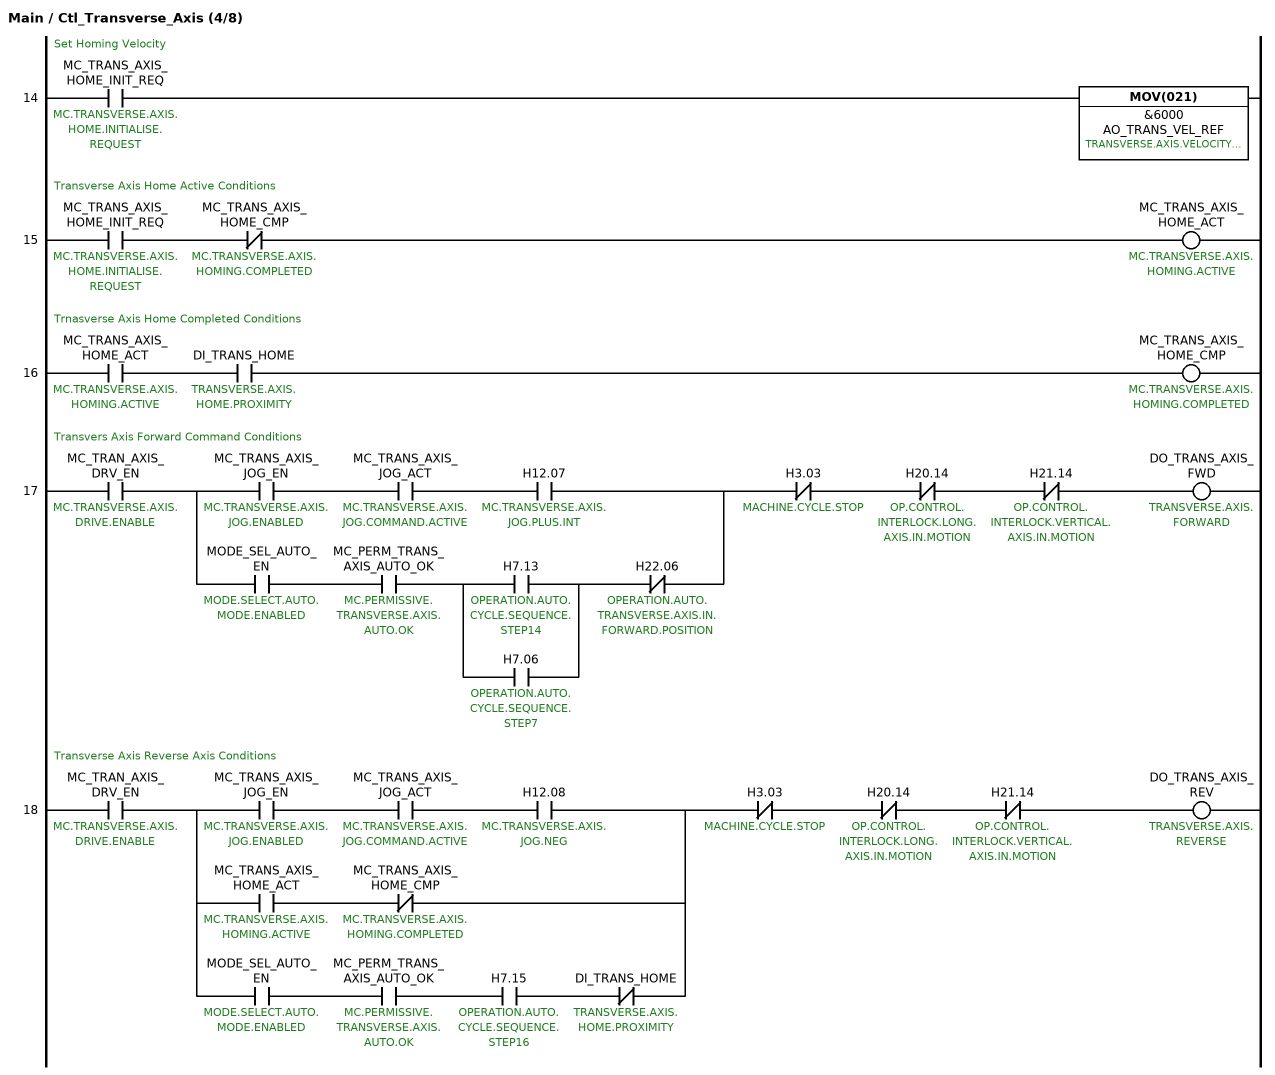
; [picture p48: Main / Ctl_Transverse_Axis, rungs 14-18]
; rung 14: Set Homing Velocity
LD MC_TRANS_AXIS_HOME_INIT_REQ  ; MC.TRANSVERSE.AXIS.HOME.INITIALISE.REQUEST
MOV(021) &6000 AO_TRANS_VEL_REF  ; TRANSVERSE.AXIS.VELOCITY.ANALOG.REFERENCE
; rung 15: Transverse Axis Home Active Conditions
LD MC_TRANS_AXIS_HOME_INIT_REQ  ; MC.TRANSVERSE.AXIS.HOME.INITIALISE.REQUEST
ANDNOT MC_TRANS_AXIS_HOME_CMP  ; MC.TRANSVERSE.AXIS.HOMING.COMPLETED
OUT MC_TRANS_AXIS_HOME_ACT  ; MC.TRANSVERSE.AXIS.HOMING.ACTIVE
; rung 16: Trnasverse Axis Home Completed Conditions
LD MC_TRANS_AXIS_HOME_ACT  ; MC.TRANSVERSE.AXIS.HOMING.ACTIVE
AND DI_TRANS_HOME  ; TRANSVERSE.AXIS.HOME.PROXIMITY
OUT MC_TRANS_AXIS_HOME_CMP  ; MC.TRANSVERSE.AXIS.HOMING.COMPLETED
; rung 17: Transvers Axis Forward Command Conditions
LD MC_TRAN_AXIS_DRV_EN  ; MC.TRANSVERSE.AXIS.DRIVE.ENABLE
LD MC_TRANS_AXIS_JOG_EN  ; MC.TRANSVERSE.AXIS.JOG.ENABLED
AND MC_TRANS_AXIS_JOG_ACT  ; MC.TRANSVERSE.AXIS.JOG.COMMAND.ACTIVE
AND H12.07  ; MC.TRANSVERSE.AXIS.JOG.PLUS.INT
LD MODE_SEL_AUTO_EN  ; MODE.SELECT.AUTO.MODE.ENABLED
AND MC_PERM_TRANS_AXIS_AUTO_OK  ; MC.PERMISSIVE.TRANSVERSE.AXIS.AUTO.OK
LD H7.13  ; OPERATION.AUTO.CYCLE.SEQUENCE.STEP14
OR H7.06  ; OPERATION.AUTO.CYCLE.SEQUENCE.STEP7
ANDLD
ANDNOT H22.06  ; OPERATION.AUTO.TRANSVERSE.AXIS.IN.FORWARD.POSITION
ORLD
ANDLD
ANDNOT H3.03  ; MACHINE.CYCLE.STOP
ANDNOT H20.14  ; OP.CONTROL.INTERLOCK.LONG.AXIS.IN.MOTION
ANDNOT H21.14  ; OP.CONTROL.INTERLOCK.VERTICAL.AXIS.IN.MOTION
OUT DO_TRANS_AXIS_FWD  ; TRANSVERSE.AXIS.FORWARD
; rung 18: Transverse Axis Reverse Axis Conditions
LD MC_TRAN_AXIS_DRV_EN  ; MC.TRANSVERSE.AXIS.DRIVE.ENABLE
LD MC_TRANS_AXIS_JOG_EN  ; MC.TRANSVERSE.AXIS.JOG.ENABLED
AND MC_TRANS_AXIS_JOG_ACT  ; MC.TRANSVERSE.AXIS.JOG.COMMAND.ACTIVE
AND H12.08  ; MC.TRANSVERSE.AXIS.JOG.NEG
LD MC_TRANS_AXIS_HOME_ACT  ; MC.TRANSVERSE.AXIS.HOMING.ACTIVE
ANDNOT MC_TRANS_AXIS_HOME_CMP  ; MC.TRANSVERSE.AXIS.HOMING.COMPLETED
ORLD
LD MODE_SEL_AUTO_EN  ; MODE.SELECT.AUTO.MODE.ENABLED
AND MC_PERM_TRANS_AXIS_AUTO_OK  ; MC.PERMISSIVE.TRANSVERSE.AXIS.AUTO.OK
AND H7.15  ; OPERATION.AUTO.CYCLE.SEQUENCE.STEP16
ANDNOT DI_TRANS_HOME  ; TRANSVERSE.AXIS.HOME.PROXIMITY
ORLD
ANDLD
ANDNOT H3.03  ; MACHINE.CYCLE.STOP
ANDNOT H20.14  ; OP.CONTROL.INTERLOCK.LONG.AXIS.IN.MOTION
ANDNOT H21.14  ; OP.CONTROL.INTERLOCK.VERTICAL.AXIS.IN.MOTION
OUT DO_TRANS_AXIS_REV  ; TRANSVERSE.AXIS.REVERSE

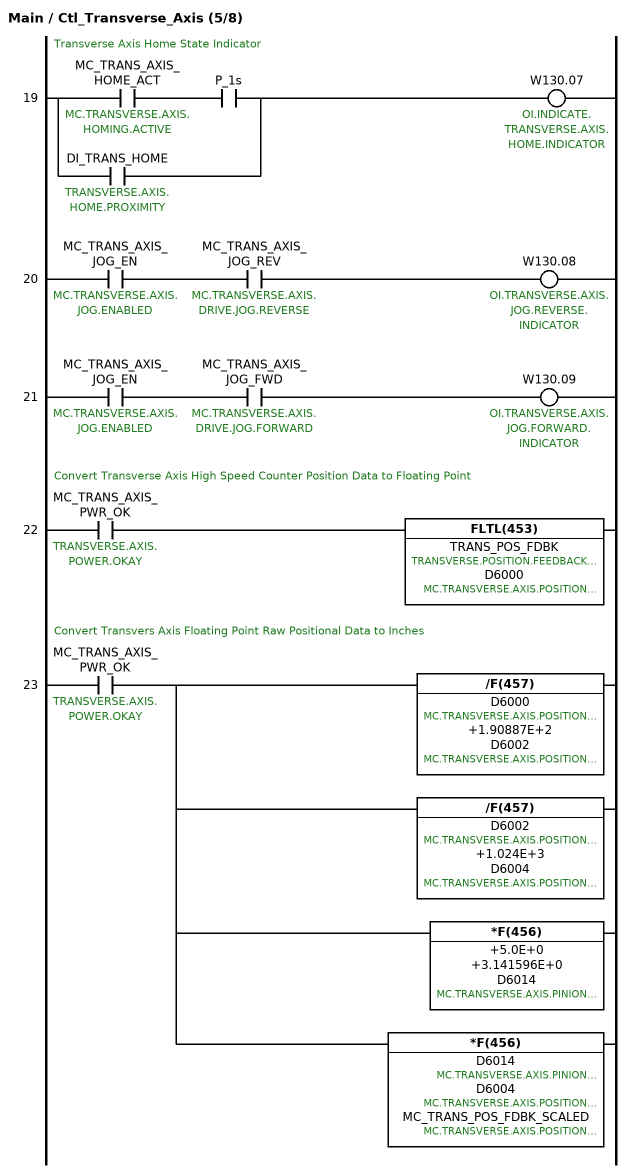
; rung 19: Transverse Axis Home State Indicator
LD MC_TRANS_AXIS_HOME_ACT  ; MC.TRANSVERSE.AXIS.HOMING.ACTIVE
AND P_1s
OR DI_TRANS_HOME  ; TRANSVERSE.AXIS.HOME.PROXIMITY
OUT W130.07  ; OI.INDICATE.TRANSVERSE.AXIS.HOME.INDICATOR
; rung 20
LD MC_TRANS_AXIS_JOG_EN  ; MC.TRANSVERSE.AXIS.JOG.ENABLED
AND MC_TRANS_AXIS_JOG_REV  ; MC.TRANSVERSE.AXIS.DRIVE.JOG.REVERSE
OUT W130.08  ; OI.TRANSVERSE.AXIS.JOG.REVERSE.INDICATOR
; rung 21
LD MC_TRANS_AXIS_JOG_EN  ; MC.TRANSVERSE.AXIS.JOG.ENABLED
AND MC_TRANS_AXIS_JOG_FWD  ; MC.TRANSVERSE.AXIS.DRIVE.JOG.FORWARD
OUT W130.09  ; OI.TRANSVERSE.AXIS.JOG.FORWARD.INDICATOR
; rung 22: Convert Transverse Axis High Speed Counter Position Data to Floating Point
LD MC_TRANS_AXIS_PWR_OK  ; TRANSVERSE.AXIS.POWER.OKAY
FLTL(453) TRANS_POS_FDBK D6000  ; TRANSVERSE.POSITION.FEEDBACK.RAW, MC.TRANSVERSE.AXIS.POSITION.FEEDBACK.RAW.REAL
; rung 23: Convert Transvers Axis Floating Point Raw Positional Data to Inches
LD MC_TRANS_AXIS_PWR_OK  ; TRANSVERSE.AXIS.POWER.OKAY
/F(457) D6000 +1.90887E+2 D6002  ; MC.TRANSVERSE.AXIS.POSITION.FEEDBACK.RAW.REAL, MC.TRANSVERSE.AXIS.POSITION.FEEDBACK.GB.SCALED.REAL
/F(457) D6002 +1.024E+3 D6004  ; MC.TRANSVERSE.AXIS.POSITION.FEEDBACK.GB.SCALED.REAL, MC.TRANSVERSE.AXIS.POSITION.PINION.REVOLUTIONS.REAL
*F(456) +5.0E+0 +3.141596E+0 D6014  ; MC.TRANSVERSE.AXIS.PINION.CIRCUMFERENCE.INCHES.REAL
*F(456) D6014 D6004 MC_TRANS_POS_FDBK_SCALED  ; MC.TRANSVERSE.AXIS.PINION.CIRCUMFERENCE.INCHES.REAL, MC.TRANSVERSE.AXIS.POSITION.PINION.REVOLUTIONS.REAL, MC.TRANSVERSE.AXIS.POSITION.FEEDBACK.INCHES.SCALED.REAL

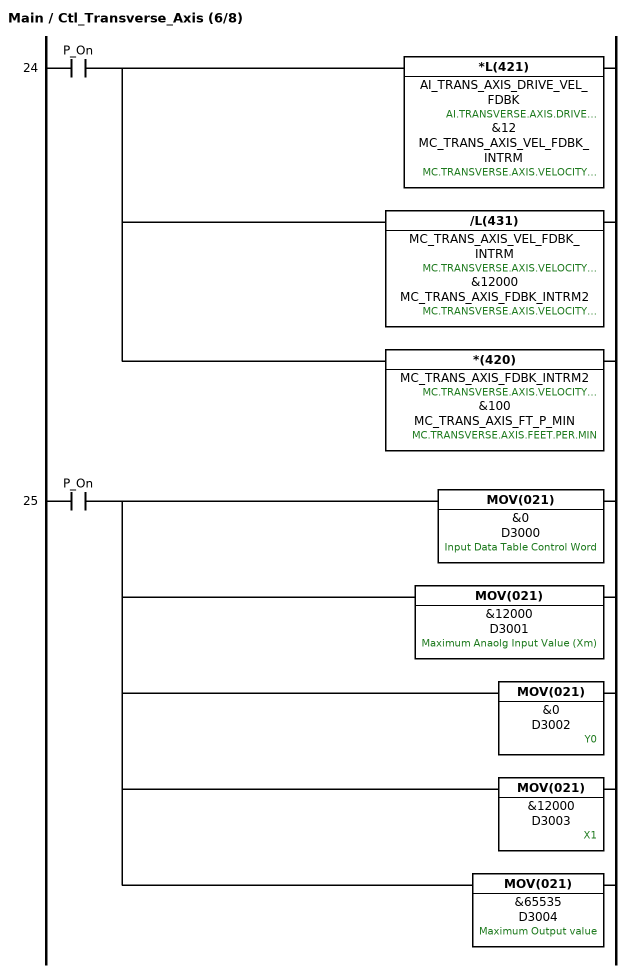
; rung 24
LD P_On
*L(421) AI_TRANS_AXIS_DRIVE_VEL_FDBK &12 MC_TRANS_AXIS_VEL_FDBK_INTRM  ; AI.TRANSVERSE.AXIS.DRIVE.VELOCITY.FEEDBACK, MC.TRANSVERSE.AXIS.VELOCITY.FEEDBACK.INTERIM
/L(431) MC_TRANS_AXIS_VEL_FDBK_INTRM &12000 MC_TRANS_AXIS_FDBK_INTRM2  ; MC.TRANSVERSE.AXIS.VELOCITY.FEEDBACK.INTERIM, MC.TRANSVERSE.AXIS.VELOCITY.FEEDBACK.INTERIM2
*(420) MC_TRANS_AXIS_FDBK_INTRM2 &100 MC_TRANS_AXIS_FT_P_MIN  ; MC.TRANSVERSE.AXIS.VELOCITY.FEEDBACK.INTERIM2, MC.TRANSVERSE.AXIS.FEET.PER.MIN
; rung 25
LD P_On
MOV(021) &0 D3000  ; Input Data Table Control Word
MOV(021) &12000 D3001  ; Maximum Anaolg Input Value (Xm)
MOV(021) &0 D3002  ; Y0
MOV(021) &12000 D3003  ; X1
MOV(021) &65535 D3004  ; Maximum Output value

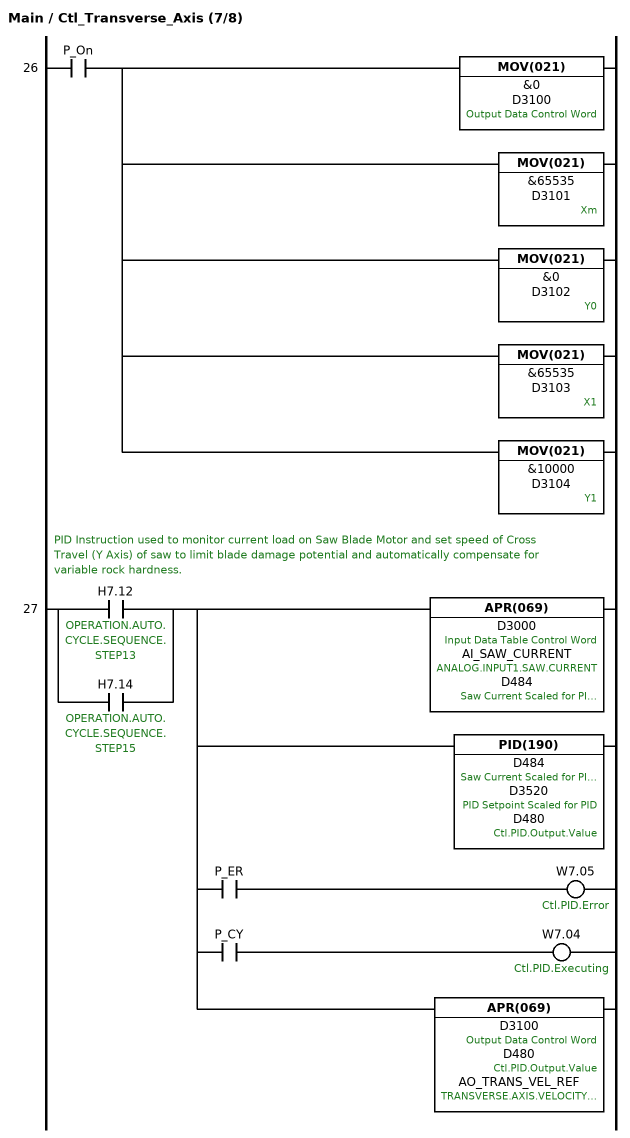
; rung 26
LD P_On
MOV(021) &0 D3100  ; Output Data Control Word
MOV(021) &65535 D3101  ; Xm
MOV(021) &0 D3102  ; Y0
MOV(021) &65535 D3103  ; X1
MOV(021) &10000 D3104  ; Y1
; rung 27: PID Instruction used to monitor current load on Saw Blade Motor and set speed of Cross Travel (Y Axis) of saw to limit blade damage potential and automatically compensate for variable rock hardness.
LD H7.12  ; OPERATION.AUTO.CYCLE.SEQUENCE.STEP13
OR H7.14  ; OPERATION.AUTO.CYCLE.SEQUENCE.STEP15
OUT TR0
APR(069) D3000 AI_SAW_CURRENT D484  ; Input Data Table Control Word, ANALOG.INPUT1.SAW.CURRENT, Saw Current Scaled for PID instruction use
PID(190) D484 D3520 D480  ; Saw Current Scaled for PID instruction use, PID Setpoint Scaled for PID, Ctl.PID.Output.Value
AND P_ER
OUT W7.05  ; Ctl.PID.Error  // Set BitW7.05 to High if PID instruction Errors
LD TR0
AND P_CY
OUT W7.04  ; Ctl.PID.Executing  // When PID is executing W7.04 is High
LD TR0
APR(069) D3100 D480 AO_TRANS_VEL_REF  ; Output Data Control Word, Ctl.PID.Output.Value, TRANSVERSE.AXIS.VELOCITY.ANALOG.REFERENCE

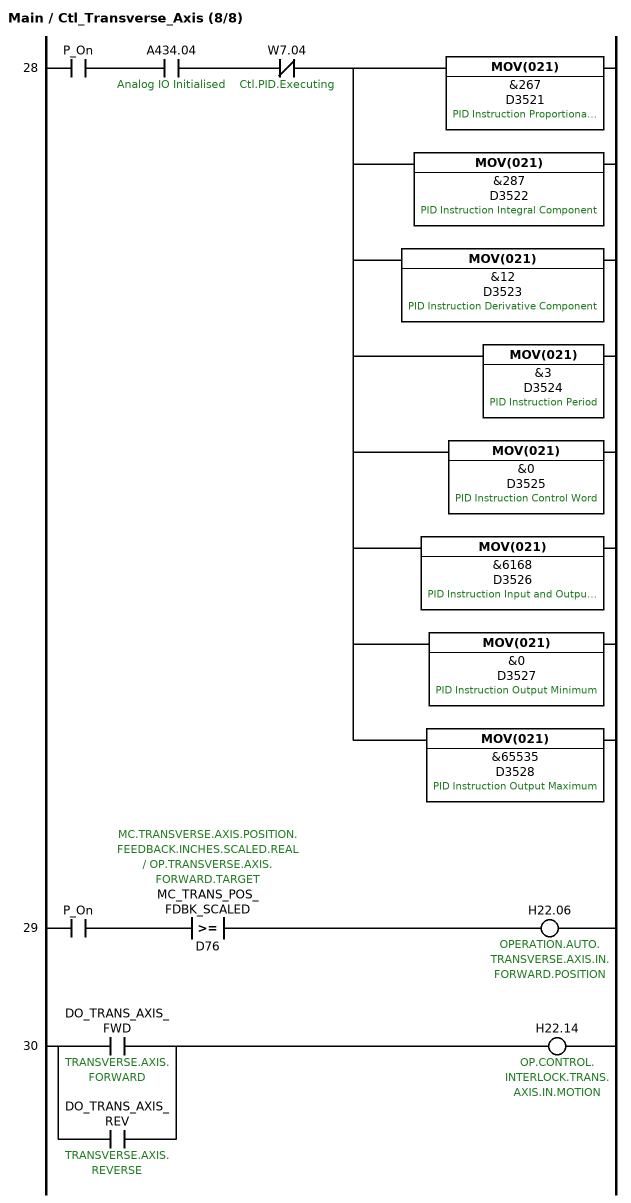
; rung 28
LD P_On
AND A434.04  ; Analog IO Initialised
ANDNOT W7.04  ; Ctl.PID.Executing
MOV(021) &267 D3521  ; PID Instruction Proportional Component
MOV(021) &287 D3522  ; PID Instruction Integral Component
MOV(021) &12 D3523  ; PID Instruction Derivative Component
MOV(021) &3 D3524  ; PID Instruction Period
MOV(021) &0 D3525  ; PID Instruction Control Word
MOV(021) &6168 D3526  ; PID Instruction Input and Output Range Setting
MOV(021) &0 D3527  ; PID Instruction Output Minimum
MOV(021) &65535 D3528  ; PID Instruction Output Maximum
; rung 29
LD P_On
AND>=F(334) MC_TRANS_POS_FDBK_SCALED D76  ; MC.TRANSVERSE.AXIS.POSITION.FEEDBACK.INCHES.SCALED.REAL, OP.TRANSVERSE.AXIS.FORWARD.TARGET
OUT H22.06  ; OPERATION.AUTO.TRANSVERSE.AXIS.IN.FORWARD.POSITION
; rung 30
LD DO_TRANS_AXIS_FWD  ; TRANSVERSE.AXIS.FORWARD
OR DO_TRANS_AXIS_REV  ; TRANSVERSE.AXIS.REVERSE
OUT H22.14  ; OP.CONTROL.INTERLOCK.TRANS.AXIS.IN.MOTION

### Section Ctl_Saw

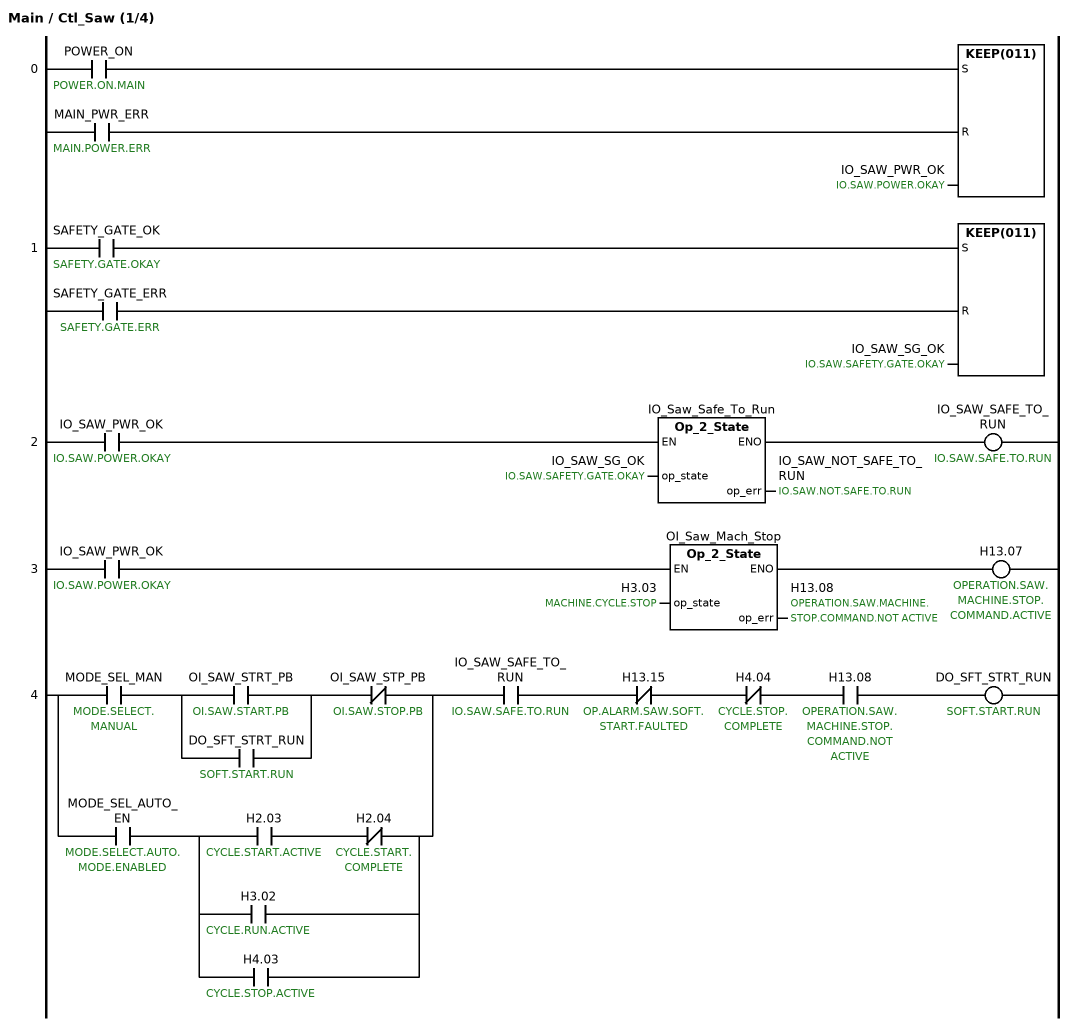
; rung 0
LD POWER_ON  ; POWER.ON.MAIN
LD MAIN_PWR_ERR  ; MAIN.POWER.ERR
KEEP(011) IO_SAW_PWR_OK  ; IO.SAW.POWER.OKAY
; rung 1
LD SAFETY_GATE_OK  ; SAFETY.GATE.OKAY
LD SAFETY_GATE_ERR  ; SAFETY.GATE.ERR
KEEP(011) IO_SAW_SG_OK  ; IO.SAW.SAFETY.GATE.OKAY
; rung 2
LD IO_SAW_PWR_OK  ; IO.SAW.POWER.OKAY
CALL IO_Saw_Safe_To_Run : Op_2_State (op_state := IO_SAW_SG_OK, op_err => IO_SAW_NOT_SAFE_TO_RUN)  ; IO.SAW.SAFETY.GATE.OKAY, IO.SAW.NOT.SAFE.TO.RUN
OUT IO_SAW_SAFE_TO_RUN  ; IO.SAW.SAFE.TO.RUN
; rung 3
LD IO_SAW_PWR_OK  ; IO.SAW.POWER.OKAY
CALL OI_Saw_Mach_Stop : Op_2_State (op_state := H3.03, op_err => H13.08)  ; MACHINE.CYCLE.STOP, OPERATION.SAW.MACHINE.STOP.COMMAND.NOT ACTIVE
OUT H13.07  ; OPERATION.SAW.MACHINE.STOP.COMMAND.ACTIVE
; rung 4
LD MODE_SEL_MAN  ; MODE.SELECT.MANUAL
LD OI_SAW_STRT_PB  ; OI.SAW.START.PB
OR DO_SFT_STRT_RUN  ; SOFT.START.RUN
ANDLD
ANDNOT OI_SAW_STP_PB  ; OI.SAW.STOP.PB
LD MODE_SEL_AUTO_EN  ; MODE.SELECT.AUTO.MODE.ENABLED
LD H2.03  ; CYCLE.START.ACTIVE
ANDNOT H2.04  ; CYCLE.START.COMPLETE
OR H3.02  ; CYCLE.RUN.ACTIVE
OR H4.03  ; CYCLE.STOP.ACTIVE
ANDLD
ORLD
AND IO_SAW_SAFE_TO_RUN  ; IO.SAW.SAFE.TO.RUN
ANDNOT H13.15  ; OP.ALARM.SAW.SOFT.START.FAULTED
ANDNOT H4.04  ; CYCLE.STOP.COMPLETE
AND H13.08  ; OPERATION.SAW.MACHINE.STOP.COMMAND.NOT ACTIVE
OUT DO_SFT_STRT_RUN  ; SOFT.START.RUN

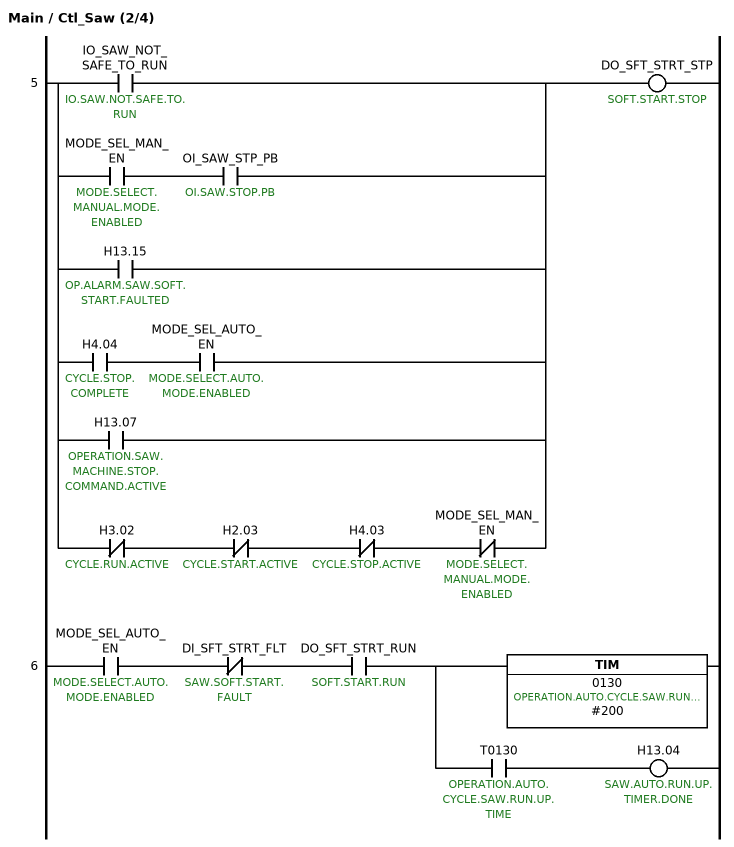
; rung 5
LD IO_SAW_NOT_SAFE_TO_RUN  ; IO.SAW.NOT.SAFE.TO.RUN
LD MODE_SEL_MAN_EN  ; MODE.SELECT.MANUAL.MODE.ENABLED
AND OI_SAW_STP_PB  ; OI.SAW.STOP.PB
ORLD
OR H13.15  ; OP.ALARM.SAW.SOFT.START.FAULTED
LD H4.04  ; CYCLE.STOP.COMPLETE
AND MODE_SEL_AUTO_EN  ; MODE.SELECT.AUTO.MODE.ENABLED
ORLD
OR H13.07  ; OPERATION.SAW.MACHINE.STOP.COMMAND.ACTIVE
LDNOT H3.02  ; CYCLE.RUN.ACTIVE
ANDNOT H2.03  ; CYCLE.START.ACTIVE
ANDNOT H4.03  ; CYCLE.STOP.ACTIVE
ANDNOT MODE_SEL_MAN_EN  ; MODE.SELECT.MANUAL.MODE.ENABLED
ORLD
OUT DO_SFT_STRT_STP  ; SOFT.START.STOP
; rung 6
LD MODE_SEL_AUTO_EN  ; MODE.SELECT.AUTO.MODE.ENABLED
ANDNOT DI_SFT_STRT_FLT  ; SAW.SOFT.START.FAULT
AND DO_SFT_STRT_RUN  ; SOFT.START.RUN
TIM 0130 #200  ; OPERATION.AUTO.CYCLE.SAW.RUN.UP.TIME
AND T0130  ; OPERATION.AUTO.CYCLE.SAW.RUN.UP.TIME
OUT H13.04  ; SAW.AUTO.RUN.UP.TIMER.DONE

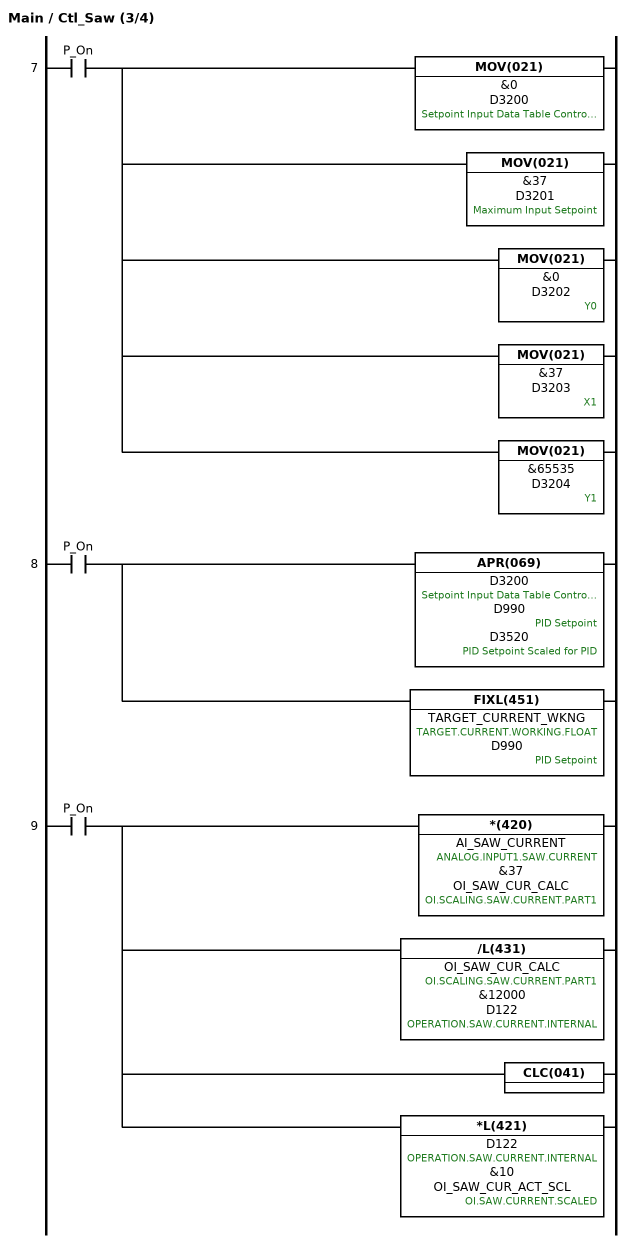
; rung 7
LD P_On
MOV(021) &0 D3200  ; Setpoint Input Data Table Control Word
MOV(021) &37 D3201  ; Maximum Input Setpoint
MOV(021) &0 D3202  ; Y0
MOV(021) &37 D3203  ; X1
MOV(021) &65535 D3204  ; Y1
; rung 8
LD P_On
APR(069) D3200 D990 D3520  ; Setpoint Input Data Table Control Word, PID Setpoint, PID Setpoint Scaled for PID
FIXL(451) TARGET_CURRENT_WKNG D990  ; TARGET.CURRENT.WORKING.FLOAT, PID Setpoint
; rung 9
LD P_On
*(420) AI_SAW_CURRENT &37 OI_SAW_CUR_CALC  ; ANALOG.INPUT1.SAW.CURRENT, OI.SCALING.SAW.CURRENT.PART1
/L(431) OI_SAW_CUR_CALC &12000 D122  ; OI.SCALING.SAW.CURRENT.PART1, OPERATION.SAW.CURRENT.INTERNAL
CLC(041)
*L(421) D122 &10 OI_SAW_CUR_ACT_SCL  ; OPERATION.SAW.CURRENT.INTERNAL, OI.SAW.CURRENT.SCALED

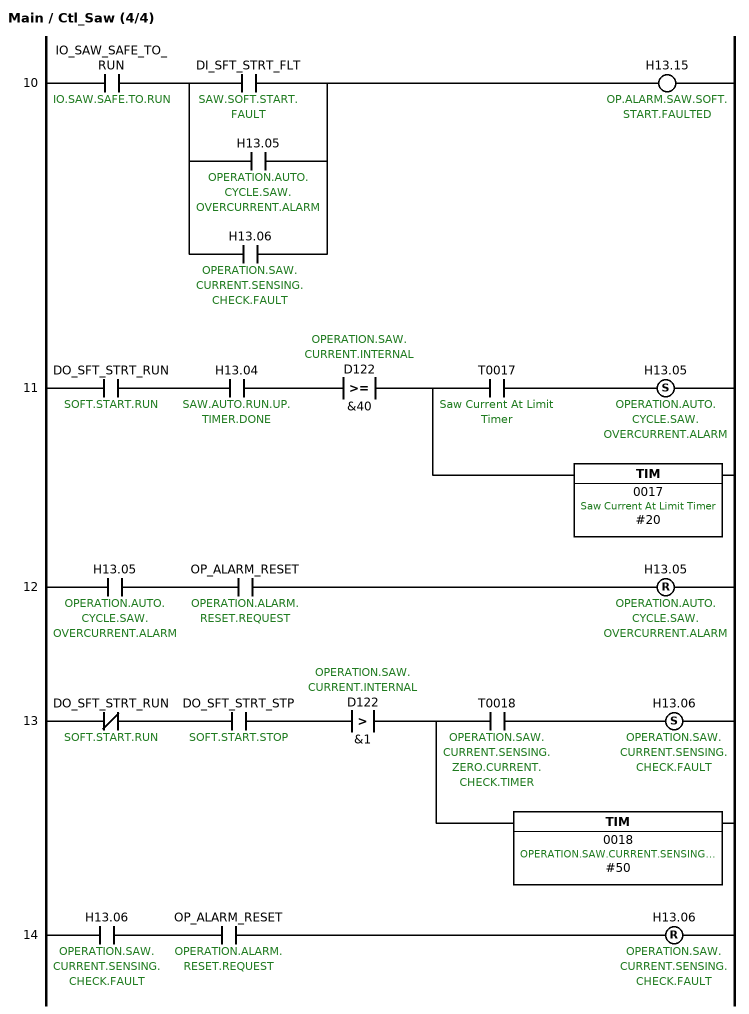
; rung 10
LD IO_SAW_SAFE_TO_RUN  ; IO.SAW.SAFE.TO.RUN
LD DI_SFT_STRT_FLT  ; SAW.SOFT.START.FAULT
OR H13.05  ; OPERATION.AUTO.CYCLE.SAW.OVERCURRENT.ALARM
OR H13.06  ; OPERATION.SAW.CURRENT.SENSING.CHECK.FAULT
ANDLD
OUT H13.15  ; OP.ALARM.SAW.SOFT.START.FAULTED
; rung 11
LD DO_SFT_STRT_RUN  ; SOFT.START.RUN
AND H13.04  ; SAW.AUTO.RUN.UP.TIMER.DONE
AND>=(325) D122 &40  ; OPERATION.SAW.CURRENT.INTERNAL
OUT TR0
AND T0017  ; Saw Current At Limit Timer
SET H13.05  ; OPERATION.AUTO.CYCLE.SAW.OVERCURRENT.ALARM
LD TR0
TIM 0017 #20  ; Saw Current At Limit Timer
; rung 12
LD H13.05  ; OPERATION.AUTO.CYCLE.SAW.OVERCURRENT.ALARM
AND OP_ALARM_RESET  ; OPERATION.ALARM.RESET.REQUEST
RSET H13.05  ; OPERATION.AUTO.CYCLE.SAW.OVERCURRENT.ALARM
; rung 13
LDNOT DO_SFT_STRT_RUN  ; SOFT.START.RUN
AND DO_SFT_STRT_STP  ; SOFT.START.STOP
AND>(320) D122 &1  ; OPERATION.SAW.CURRENT.INTERNAL
OUT TR0
AND T0018  ; OPERATION.SAW.CURRENT.SENSING.ZERO.CURRENT.CHECK.TIMER
SET H13.06  ; OPERATION.SAW.CURRENT.SENSING.CHECK.FAULT
LD TR0
TIM 0018 #50  ; OPERATION.SAW.CURRENT.SENSING.ZERO.CURRENT.CHECK.TIMER
; rung 14
LD H13.06  ; OPERATION.SAW.CURRENT.SENSING.CHECK.FAULT
AND OP_ALARM_RESET  ; OPERATION.ALARM.RESET.REQUEST
RSET H13.06  ; OPERATION.SAW.CURRENT.SENSING.CHECK.FAULT

### Section Ctl_Water

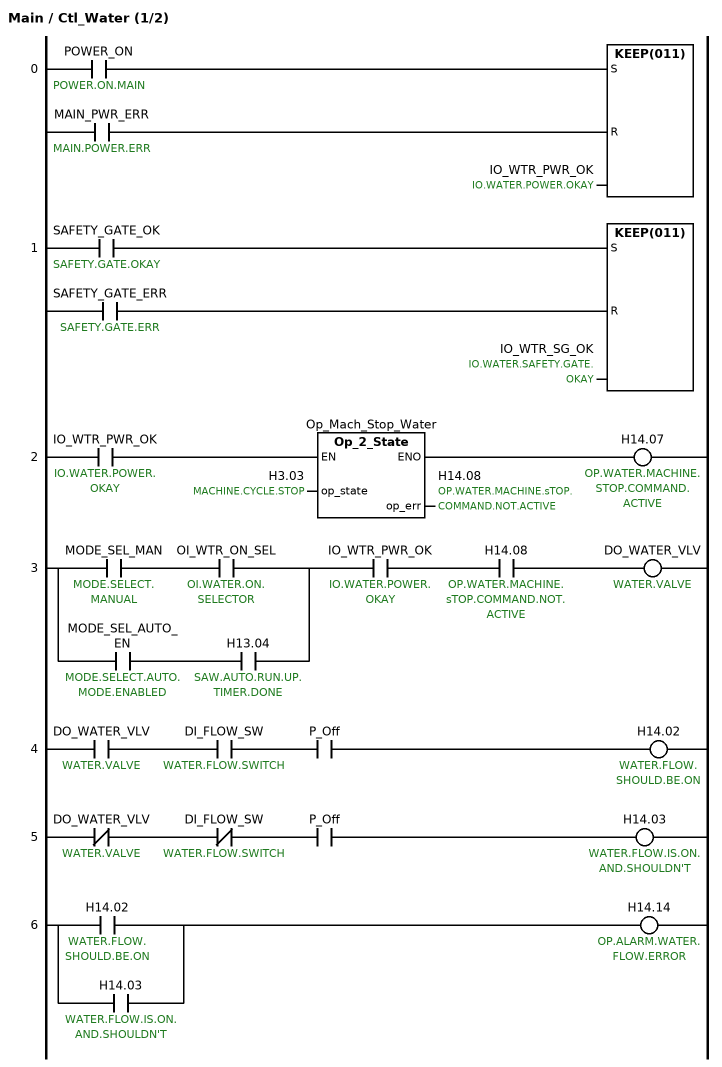
; rung 0
LD POWER_ON  ; POWER.ON.MAIN
LD MAIN_PWR_ERR  ; MAIN.POWER.ERR
KEEP(011) IO_WTR_PWR_OK  ; IO.WATER.POWER.OKAY
; rung 1
LD SAFETY_GATE_OK  ; SAFETY.GATE.OKAY
LD SAFETY_GATE_ERR  ; SAFETY.GATE.ERR
KEEP(011) IO_WTR_SG_OK  ; IO.WATER.SAFETY.GATE.OKAY
; rung 2
LD IO_WTR_PWR_OK  ; IO.WATER.POWER.OKAY
CALL Op_Mach_Stop_Water : Op_2_State (op_state := H3.03, op_err => H14.08)  ; MACHINE.CYCLE.STOP, OP.WATER.MACHINE.sTOP.COMMAND.NOT.ACTIVE
OUT H14.07  ; OP.WATER.MACHINE.STOP.COMMAND.ACTIVE
; rung 3
LD MODE_SEL_MAN  ; MODE.SELECT.MANUAL
AND OI_WTR_ON_SEL  ; OI.WATER.ON.SELECTOR
LD MODE_SEL_AUTO_EN  ; MODE.SELECT.AUTO.MODE.ENABLED
AND H13.04  ; SAW.AUTO.RUN.UP.TIMER.DONE
ORLD
AND IO_WTR_PWR_OK  ; IO.WATER.POWER.OKAY
AND H14.08  ; OP.WATER.MACHINE.sTOP.COMMAND.NOT.ACTIVE
OUT DO_WATER_VLV  ; WATER.VALVE
; rung 4
LD DO_WATER_VLV  ; WATER.VALVE
AND DI_FLOW_SW  ; WATER.FLOW.SWITCH
AND P_Off
OUT H14.02  ; WATER.FLOW.SHOULD.BE.ON
; rung 5
LDNOT DO_WATER_VLV  ; WATER.VALVE
ANDNOT DI_FLOW_SW  ; WATER.FLOW.SWITCH
AND P_Off
OUT H14.03  ; WATER.FLOW.IS.ON.AND.SHOULDN'T
; rung 6
LD H14.02  ; WATER.FLOW.SHOULD.BE.ON
OR H14.03  ; WATER.FLOW.IS.ON.AND.SHOULDN'T
OUT H14.14  ; OP.ALARM.WATER.FLOW.ERROR

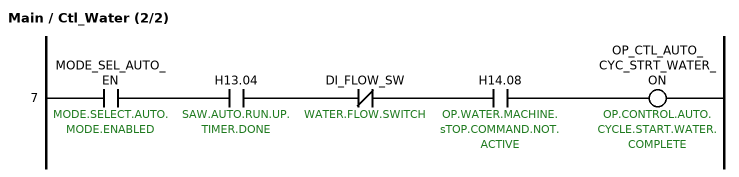
; rung 7
LD MODE_SEL_AUTO_EN  ; MODE.SELECT.AUTO.MODE.ENABLED
AND H13.04  ; SAW.AUTO.RUN.UP.TIMER.DONE
ANDNOT DI_FLOW_SW  ; WATER.FLOW.SWITCH
AND H14.08  ; OP.WATER.MACHINE.sTOP.COMMAND.NOT.ACTIVE
OUT OP_CTL_AUTO_CYC_STRT_WATER_ON  ; OP.CONTROL.AUTO.CYCLE.START.WATER.COMPLETE

### Section Ctl_Lazer

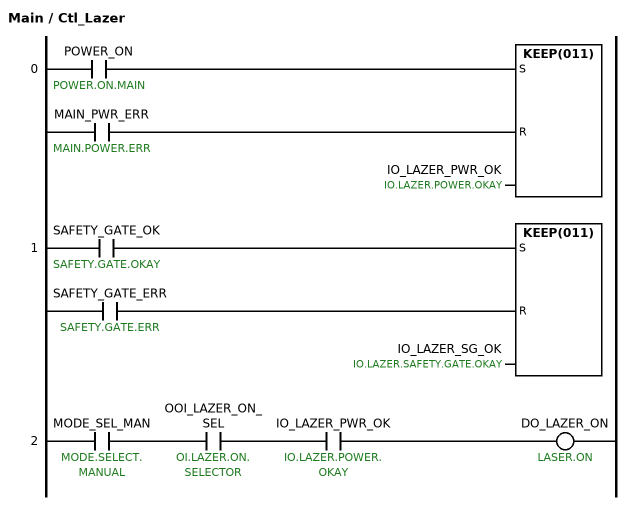
; rung 0
LD POWER_ON  ; POWER.ON.MAIN
LD MAIN_PWR_ERR  ; MAIN.POWER.ERR
KEEP(011) IO_LAZER_PWR_OK  ; IO.LAZER.POWER.OKAY
; rung 1
LD SAFETY_GATE_OK  ; SAFETY.GATE.OKAY
LD SAFETY_GATE_ERR  ; SAFETY.GATE.ERR
KEEP(011) IO_LAZER_SG_OK  ; IO.LAZER.SAFETY.GATE.OKAY
; rung 2
LD MODE_SEL_MAN  ; MODE.SELECT.MANUAL
AND OOI_LAZER_ON_SEL  ; OI.LAZER.ON.SELECTOR
AND IO_LAZER_PWR_OK  ; IO.LAZER.POWER.OKAY
OUT DO_LAZER_ON  ; LASER.ON

### Section Init_Recipe

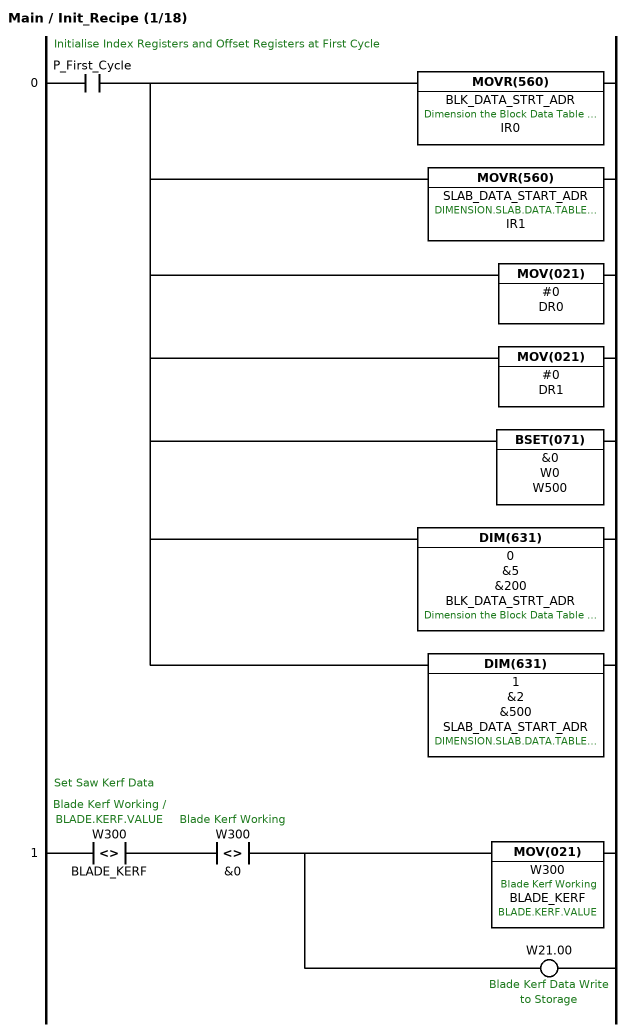
; rung 0: Initialise Index Registers and Offset Registers at First Cycle
LD P_First_Cycle
MOVR(560) BLK_DATA_STRT_ADR IR0  ; Dimension the Block Data Table - Start Address
MOVR(560) SLAB_DATA_START_ADR IR1  ; DIMENSION.SLAB.DATA.TABLE.START.ADDRESS
MOV(021) #0 DR0
MOV(021) #0 DR1
BSET(071) &0 W0 W500
DIM(631) 0 &5 &200 BLK_DATA_STRT_ADR  ; Dimension the Block Data Table - Start Address
DIM(631) 1 &2 &500 SLAB_DATA_START_ADR  ; DIMENSION.SLAB.DATA.TABLE.START.ADDRESS
; rung 1: Set Saw Kerf Data
LD<>(305) W300 BLADE_KERF  ; Blade Kerf Working, BLADE.KERF.VALUE
AND<>(305) W300 &0  ; Blade Kerf Working
MOV(021) W300 BLADE_KERF  ; Blade Kerf Working, BLADE.KERF.VALUE
OUT W21.00  ; Blade Kerf Data Write to Storage

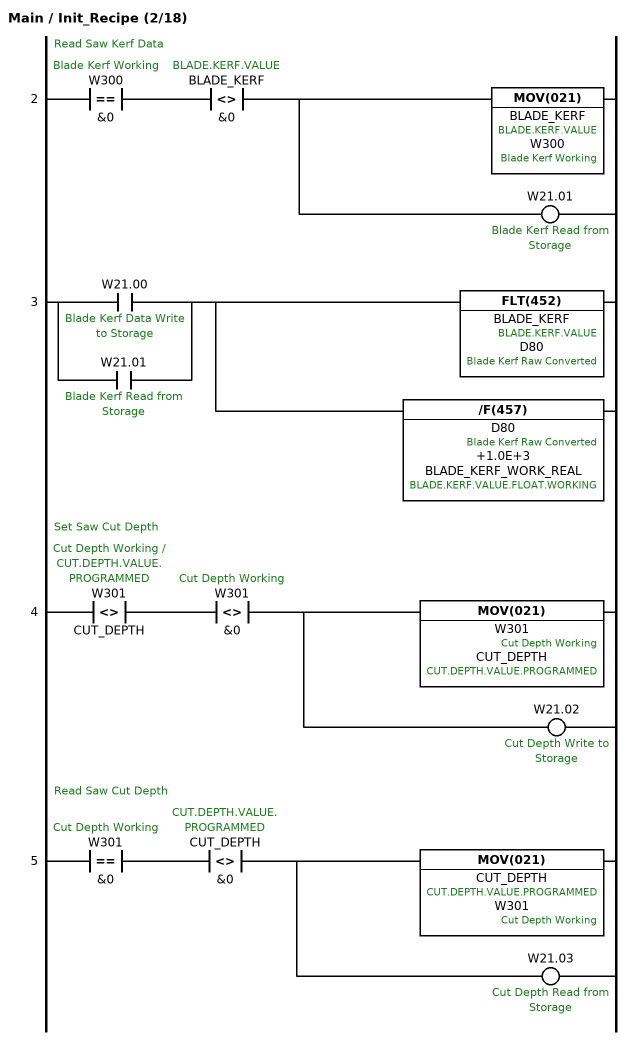
; rung 2: Read Saw Kerf Data
LD=(300) W300 &0  ; Blade Kerf Working
AND<>(305) BLADE_KERF &0  ; BLADE.KERF.VALUE
MOV(021) BLADE_KERF W300  ; BLADE.KERF.VALUE, Blade Kerf Working
OUT W21.01  ; Blade Kerf Read from Storage
; rung 3
LD W21.00  ; Blade Kerf Data Write to Storage
OR W21.01  ; Blade Kerf Read from Storage
FLT(452) BLADE_KERF D80  ; BLADE.KERF.VALUE, Blade Kerf Raw Converted
/F(457) D80 +1.0E+3 BLADE_KERF_WORK_REAL  ; Blade Kerf Raw Converted, BLADE.KERF.VALUE.FLOAT.WORKING
; rung 4: Set Saw Cut Depth
LD<>(305) W301 CUT_DEPTH  ; Cut Depth Working, CUT.DEPTH.VALUE.PROGRAMMED
AND<>(305) W301 &0  ; Cut Depth Working
MOV(021) W301 CUT_DEPTH  ; Cut Depth Working, CUT.DEPTH.VALUE.PROGRAMMED
OUT W21.02  ; Cut Depth Write to Storage
; rung 5: Read Saw Cut Depth
LD=(300) W301 &0  ; Cut Depth Working
AND<>(305) CUT_DEPTH &0  ; CUT.DEPTH.VALUE.PROGRAMMED
MOV(021) CUT_DEPTH W301  ; CUT.DEPTH.VALUE.PROGRAMMED, Cut Depth Working
OUT W21.03  ; Cut Depth Read from Storage

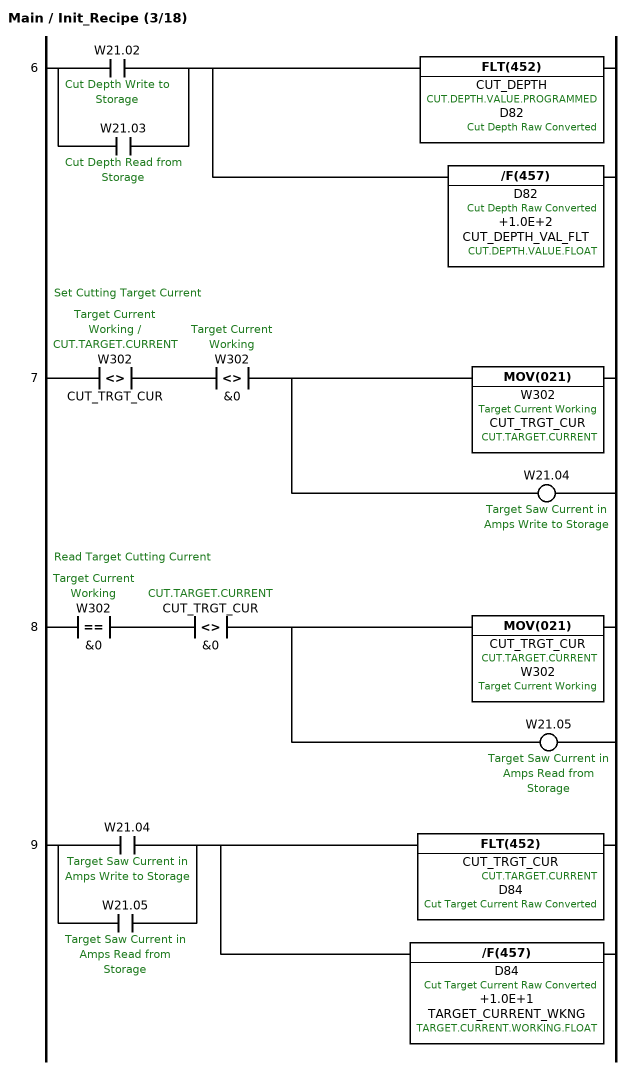
; rung 6
LD W21.02  ; Cut Depth Write to Storage
OR W21.03  ; Cut Depth Read from Storage
FLT(452) CUT_DEPTH D82  ; CUT.DEPTH.VALUE.PROGRAMMED, Cut Depth Raw Converted
/F(457) D82 +1.0E+2 CUT_DEPTH_VAL_FLT  ; Cut Depth Raw Converted, CUT.DEPTH.VALUE.FLOAT
; rung 7: Set Cutting Target Current
LD<>(305) W302 CUT_TRGT_CUR  ; Target Current Working, CUT.TARGET.CURRENT
AND<>(305) W302 &0  ; Target Current Working
MOV(021) W302 CUT_TRGT_CUR  ; Target Current Working, CUT.TARGET.CURRENT
OUT W21.04  ; Target Saw Current in Amps Write to Storage
; rung 8: Read Target Cutting Current
LD=(300) W302 &0  ; Target Current Working
AND<>(305) CUT_TRGT_CUR &0  ; CUT.TARGET.CURRENT
MOV(021) CUT_TRGT_CUR W302  ; CUT.TARGET.CURRENT, Target Current Working
OUT W21.05  ; Target Saw Current in Amps Read from Storage
; rung 9
LD W21.04  ; Target Saw Current in Amps Write to Storage
OR W21.05  ; Target Saw Current in Amps Read from Storage
FLT(452) CUT_TRGT_CUR D84  ; CUT.TARGET.CURRENT, Cut Target Current Raw Converted
/F(457) D84 +1.0E+1 TARGET_CURRENT_WKNG  ; Cut Target Current Raw Converted, TARGET.CURRENT.WORKING.FLOAT

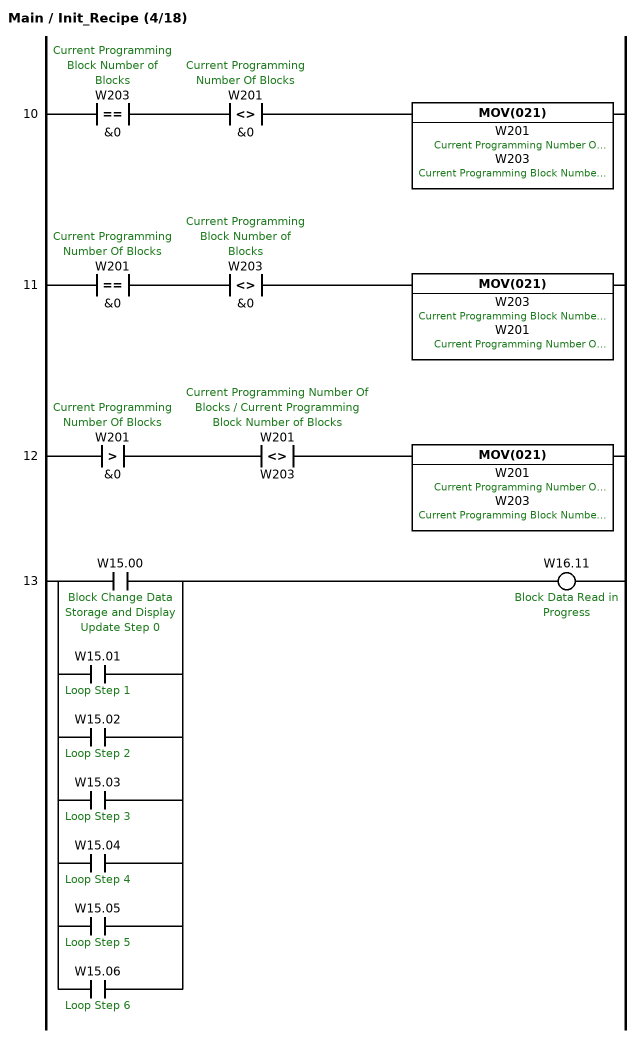
; rung 10
LD=(300) W203 &0  ; Current Programming Block Number of Blocks
AND<>(305) W201 &0  ; Current Programming Number Of Blocks
MOV(021) W201 W203  ; Current Programming Number Of Blocks, Current Programming Block Number of Blocks
; rung 11
LD=(300) W201 &0  ; Current Programming Number Of Blocks
AND<>(305) W203 &0  ; Current Programming Block Number of Blocks
MOV(021) W203 W201  ; Current Programming Block Number of Blocks, Current Programming Number Of Blocks
; rung 12
LD>(320) W201 &0  ; Current Programming Number Of Blocks
AND<>(305) W201 W203  ; Current Programming Number Of Blocks, Current Programming Block Number of Blocks
MOV(021) W201 W203  ; Current Programming Number Of Blocks, Current Programming Block Number of Blocks
; rung 13
LD W15.00  ; Block Change Data Storage and Display Update Step 0
OR W15.01  ; Loop Step 1
OR W15.02  ; Loop Step 2
OR W15.03  ; Loop Step 3
OR W15.04  ; Loop Step 4
OR W15.05  ; Loop Step 5
OR W15.06  ; Loop Step 6
OUT W16.11  ; Block Data Read in Progress

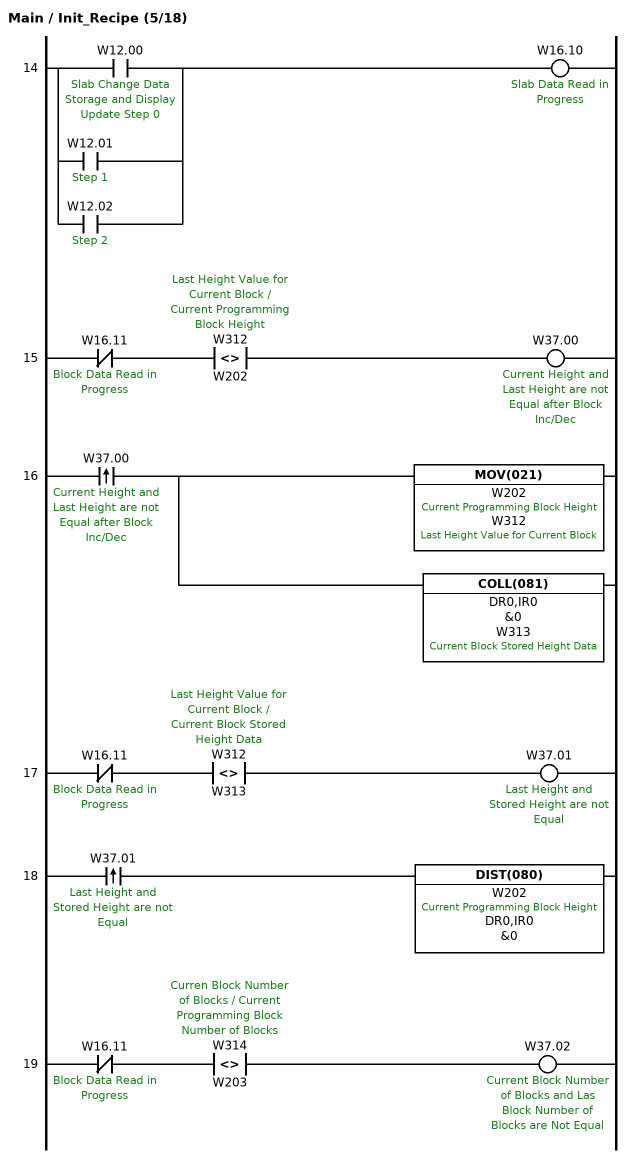
; rung 14
LD W12.00  ; Slab Change Data Storage and Display Update Step 0
OR W12.01  ; Step 1
OR W12.02  ; Step 2
OUT W16.10  ; Slab Data Read in Progress
; rung 15
LDNOT W16.11  ; Block Data Read in Progress
AND<>(305) W312 W202  ; Last Height Value for Current Block, Current Programming Block Height
OUT W37.00  ; Current Height and Last Height are not Equal after Block Inc/Dec
; rung 16
@LD W37.00  ; Current Height and Last Height are not Equal after Block Inc/Dec
MOV(021) W202 W312  ; Current Programming Block Height, Last Height Value for Current Block
COLL(081) DR0,IR0 &0 W313  ; Current Block Stored Height Data
; rung 17
LDNOT W16.11  ; Block Data Read in Progress
AND<>(305) W312 W313  ; Last Height Value for Current Block, Current Block Stored Height Data
OUT W37.01  ; Last Height and Stored Height are not Equal
; rung 18
@LD W37.01  ; Last Height and Stored Height are not Equal
DIST(080) W202 DR0,IR0 &0  ; Current Programming Block Height
; rung 19
LDNOT W16.11  ; Block Data Read in Progress
AND<>(305) W314 W203  ; Curren Block Number of Blocks, Current Programming Block Number of Blocks
OUT W37.02  ; Current Block Number of Blocks and Las Block Number of Blocks are Not Equal

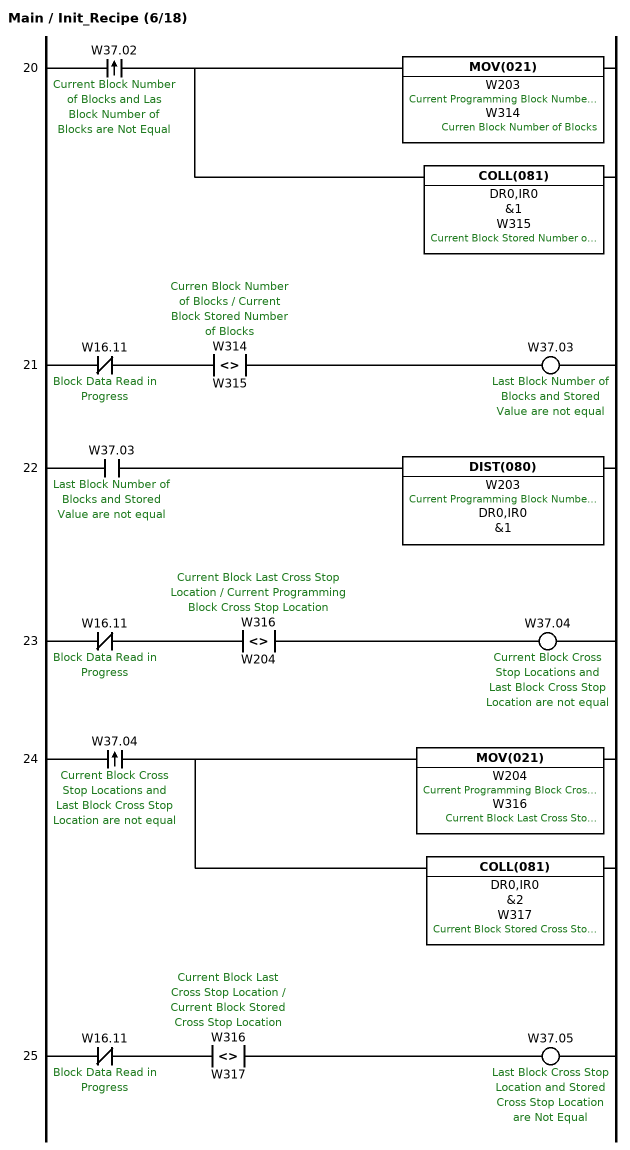
; rung 20
@LD W37.02  ; Current Block Number of Blocks and Las Block Number of Blocks are Not Equal
MOV(021) W203 W314  ; Current Programming Block Number of Blocks, Curren Block Number of Blocks
COLL(081) DR0,IR0 &1 W315  ; Current Block Stored Number of Blocks
; rung 21
LDNOT W16.11  ; Block Data Read in Progress
AND<>(305) W314 W315  ; Curren Block Number of Blocks, Current Block Stored Number of Blocks
OUT W37.03  ; Last Block Number of Blocks and Stored Value are not equal
; rung 22
LD W37.03  ; Last Block Number of Blocks and Stored Value are not equal
DIST(080) W203 DR0,IR0 &1  ; Current Programming Block Number of Blocks
; rung 23
LDNOT W16.11  ; Block Data Read in Progress
AND<>(305) W316 W204  ; Current Block Last Cross Stop Location, Current Programming Block Cross Stop Location
OUT W37.04  ; Current Block Cross Stop Locations and Last Block Cross Stop Location are not equal
; rung 24
@LD W37.04  ; Current Block Cross Stop Locations and Last Block Cross Stop Location are not equal
MOV(021) W204 W316  ; Current Programming Block Cross Stop Location, Current Block Last Cross Stop Location
COLL(081) DR0,IR0 &2 W317  ; Current Block Stored Cross Stop Location
; rung 25
LDNOT W16.11  ; Block Data Read in Progress
AND<>(305) W316 W317  ; Current Block Last Cross Stop Location, Current Block Stored Cross Stop Location
OUT W37.05  ; Last Block Cross Stop Location and Stored Cross Stop Location are Not Equal

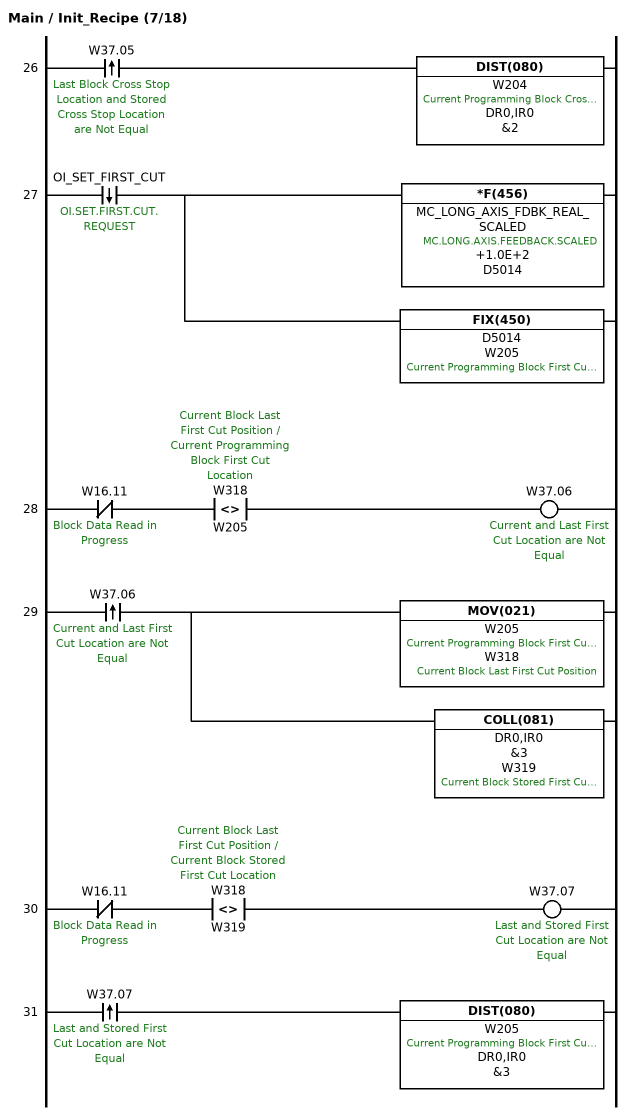
; rung 26
@LD W37.05  ; Last Block Cross Stop Location and Stored Cross Stop Location are Not Equal
DIST(080) W204 DR0,IR0 &2  ; Current Programming Block Cross Stop Location
; rung 27
%LD OI_SET_FIRST_CUT  ; OI.SET.FIRST.CUT.REQUEST
*F(456) MC_LONG_AXIS_FDBK_REAL_SCALED +1.0E+2 D5014  ; MC.LONG.AXIS.FEEDBACK.SCALED
FIX(450) D5014 W205  ; Current Programming Block First Cut Location
; rung 28
LDNOT W16.11  ; Block Data Read in Progress
AND<>(305) W318 W205  ; Current Block Last First Cut Position, Current Programming Block First Cut Location
OUT W37.06  ; Current and Last First Cut Location are Not Equal
; rung 29
@LD W37.06  ; Current and Last First Cut Location are Not Equal
MOV(021) W205 W318  ; Current Programming Block First Cut Location, Current Block Last First Cut Position
COLL(081) DR0,IR0 &3 W319  ; Current Block Stored First Cut Location
; rung 30
LDNOT W16.11  ; Block Data Read in Progress
AND<>(305) W318 W319  ; Current Block Last First Cut Position, Current Block Stored First Cut Location
OUT W37.07  ; Last and Stored First Cut Location are Not Equal
; rung 31
@LD W37.07  ; Last and Stored First Cut Location are Not Equal
DIST(080) W205 DR0,IR0 &3  ; Current Programming Block First Cut Location

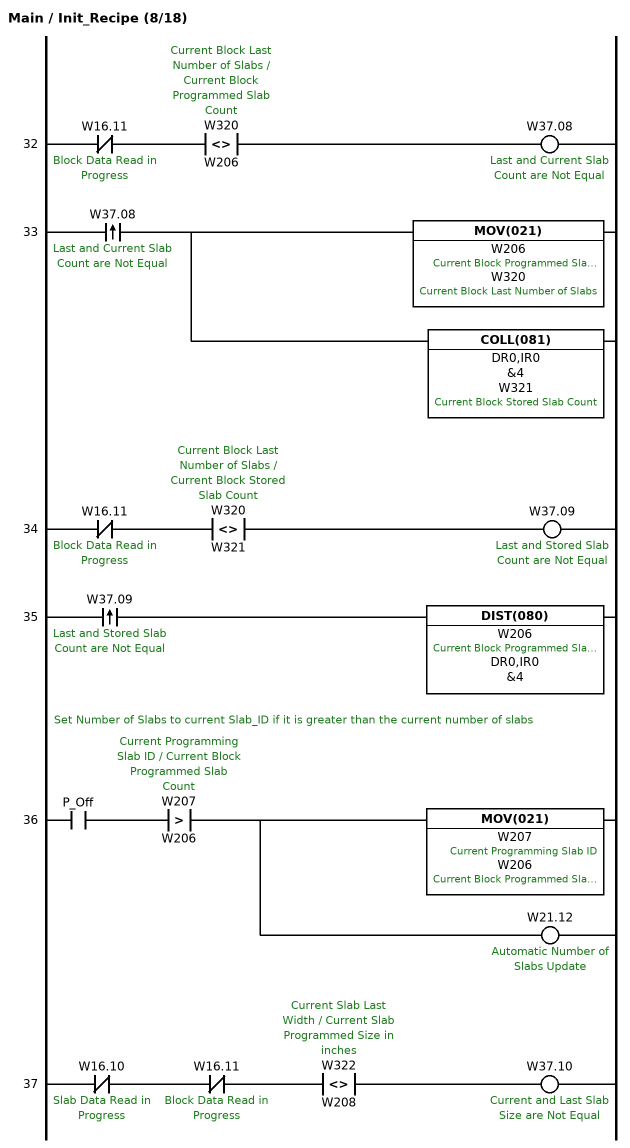
; rung 32
LDNOT W16.11  ; Block Data Read in Progress
AND<>(305) W320 W206  ; Current Block Last Number of Slabs, Current Block Programmed Slab Count
OUT W37.08  ; Last and Current Slab Count are Not Equal
; rung 33
@LD W37.08  ; Last and Current Slab Count are Not Equal
MOV(021) W206 W320  ; Current Block Programmed Slab Count, Current Block Last Number of Slabs
COLL(081) DR0,IR0 &4 W321  ; Current Block Stored Slab Count
; rung 34
LDNOT W16.11  ; Block Data Read in Progress
AND<>(305) W320 W321  ; Current Block Last Number of Slabs, Current Block Stored Slab Count
OUT W37.09  ; Last and Stored Slab Count are Not Equal
; rung 35
@LD W37.09  ; Last and Stored Slab Count are Not Equal
DIST(080) W206 DR0,IR0 &4  ; Current Block Programmed Slab Count
; rung 36: Set Number of Slabs to current Slab_ID if it is greater than the current number of slabs
LD P_Off
AND>(320) W207 W206  ; Current Programming Slab ID, Current Block Programmed Slab Count
MOV(021) W207 W206  ; Current Programming Slab ID, Current Block Programmed Slab Count
OUT W21.12  ; Automatic Number of Slabs Update
; rung 37
LDNOT W16.10  ; Slab Data Read in Progress
ANDNOT W16.11  ; Block Data Read in Progress
AND<>(305) W322 W208  ; Current Slab Last Width, Current Slab Programmed Size in inches
OUT W37.10  ; Current and Last Slab Size are Not Equal

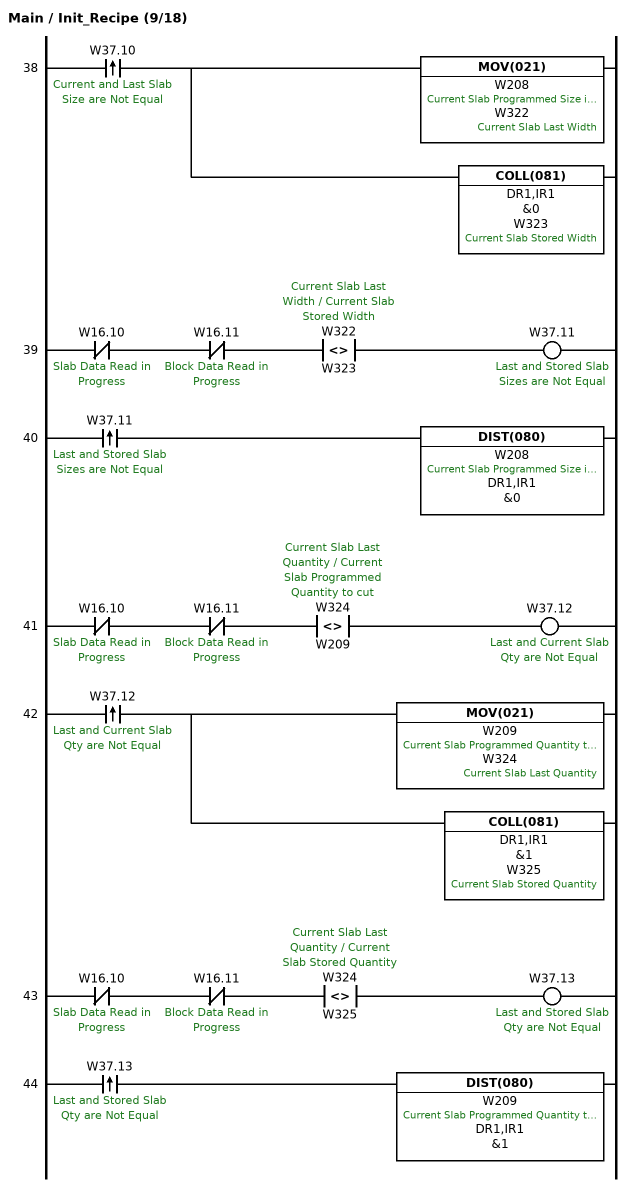
; rung 38
@LD W37.10  ; Current and Last Slab Size are Not Equal
MOV(021) W208 W322  ; Current Slab Programmed Size in inches, Current Slab Last Width
COLL(081) DR1,IR1 &0 W323  ; Current Slab Stored Width
; rung 39
LDNOT W16.10  ; Slab Data Read in Progress
ANDNOT W16.11  ; Block Data Read in Progress
AND<>(305) W322 W323  ; Current Slab Last Width, Current Slab Stored Width
OUT W37.11  ; Last and Stored Slab Sizes are Not Equal
; rung 40
@LD W37.11  ; Last and Stored Slab Sizes are Not Equal
DIST(080) W208 DR1,IR1 &0  ; Current Slab Programmed Size in inches
; rung 41
LDNOT W16.10  ; Slab Data Read in Progress
ANDNOT W16.11  ; Block Data Read in Progress
AND<>(305) W324 W209  ; Current Slab Last Quantity, Current Slab Programmed Quantity to cut
OUT W37.12  ; Last and Current Slab Qty are Not Equal
; rung 42
@LD W37.12  ; Last and Current Slab Qty are Not Equal
MOV(021) W209 W324  ; Current Slab Programmed Quantity to cut, Current Slab Last Quantity
COLL(081) DR1,IR1 &1 W325  ; Current Slab Stored Quantity
; rung 43
LDNOT W16.10  ; Slab Data Read in Progress
ANDNOT W16.11  ; Block Data Read in Progress
AND<>(305) W324 W325  ; Current Slab Last Quantity, Current Slab Stored Quantity
OUT W37.13  ; Last and Stored Slab Qty are Not Equal
; rung 44
@LD W37.13  ; Last and Stored Slab Qty are Not Equal
DIST(080) W209 DR1,IR1 &1  ; Current Slab Programmed Quantity to cut

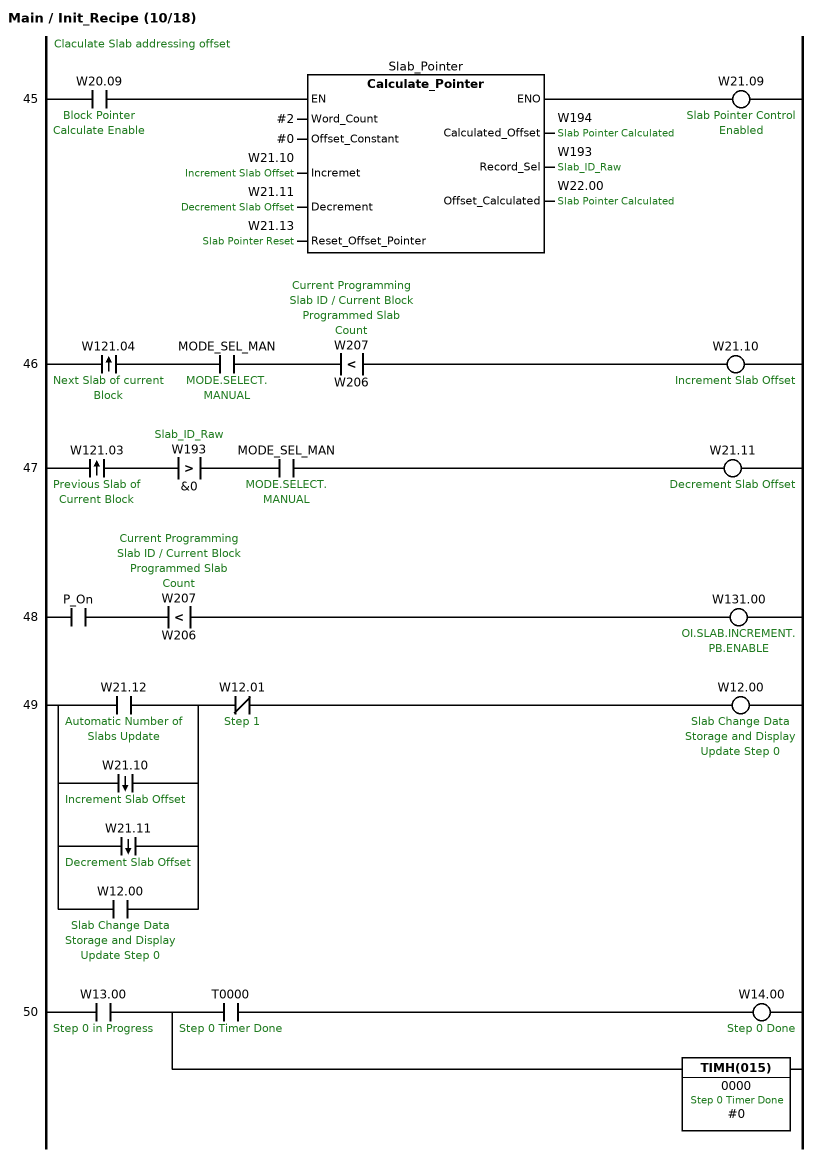
; rung 45: Claculate Slab addressing offset
LD W20.09  ; Block Pointer Calculate Enable
CALL Slab_Pointer : Calculate_Pointer (Word_Count := #2, Offset_Constant := #0, Incremet := W21.10, Decrement := W21.11, Reset_Offset_Pointer := W21.13, Calculated_Offset => W194, Record_Sel => W193, Offset_Calculated => W22.00)  ; Increment Slab Offset, Decrement Slab Offset, Slab Pointer Reset, Slab Pointer Calculated, Slab_ID_Raw
OUT W21.09  ; Slab Pointer Control Enabled
; rung 46
@LD W121.04  ; Next Slab of current Block
AND MODE_SEL_MAN  ; MODE.SELECT.MANUAL
AND<(310) W207 W206  ; Current Programming Slab ID, Current Block Programmed Slab Count
OUT W21.10  ; Increment Slab Offset
; rung 47
@LD W121.03  ; Previous Slab of Current Block
AND>(320) W193 &0  ; Slab_ID_Raw
AND MODE_SEL_MAN  ; MODE.SELECT.MANUAL
OUT W21.11  ; Decrement Slab Offset
; rung 48
LD P_On
AND<(310) W207 W206  ; Current Programming Slab ID, Current Block Programmed Slab Count
OUT W131.00  ; OI.SLAB.INCREMENT.PB.ENABLE
; rung 49
LD W21.12  ; Automatic Number of Slabs Update
%OR W21.10  ; Increment Slab Offset
%OR W21.11  ; Decrement Slab Offset
OR W12.00  ; Slab Change Data Storage and Display Update Step 0
ANDNOT W12.01  ; Step 1
OUT W12.00  ; Slab Change Data Storage and Display Update Step 0
; rung 50
LD W13.00  ; Step 0 in Progress
OUT TR0
AND T0000  ; Step 0 Timer Done
OUT W14.00  ; Step 0 Done
LD TR0
TIMH(015) 0000 #0  ; Step 0 Timer Done

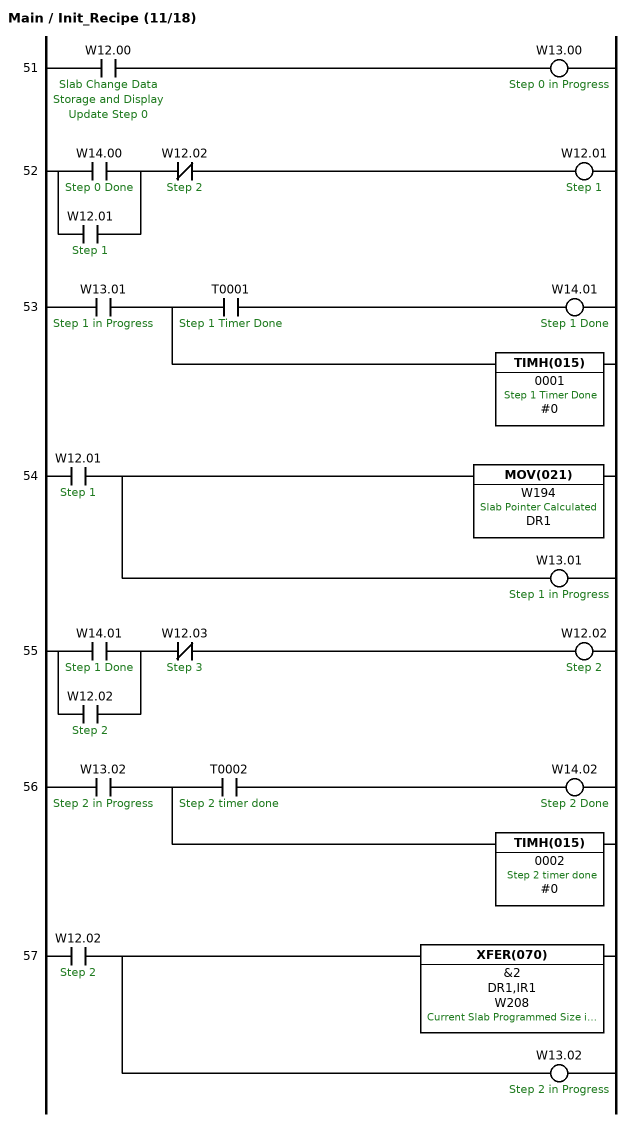
; rung 51
LD W12.00  ; Slab Change Data Storage and Display Update Step 0
OUT W13.00  ; Step 0 in Progress
; rung 52
LD W14.00  ; Step 0 Done
OR W12.01  ; Step 1
ANDNOT W12.02  ; Step 2
OUT W12.01  ; Step 1
; rung 53
LD W13.01  ; Step 1 in Progress
OUT TR0
AND T0001  ; Step 1 Timer Done
OUT W14.01  ; Step 1 Done
LD TR0
TIMH(015) 0001 #0  ; Step 1 Timer Done
; rung 54
LD W12.01  ; Step 1
MOV(021) W194 DR1  ; Slab Pointer Calculated
OUT W13.01  ; Step 1 in Progress
; rung 55
LD W14.01  ; Step 1 Done
OR W12.02  ; Step 2
ANDNOT W12.03  ; Step 3
OUT W12.02  ; Step 2
; rung 56
LD W13.02  ; Step 2 in Progress
OUT TR0
AND T0002  ; Step 2 timer done
OUT W14.02  ; Step 2 Done
LD TR0
TIMH(015) 0002 #0  ; Step 2 timer done
; rung 57
LD W12.02  ; Step 2
XFER(070) &2 DR1,IR1 W208  ; Current Slab Programmed Size in inches
OUT W13.02  ; Step 2 in Progress

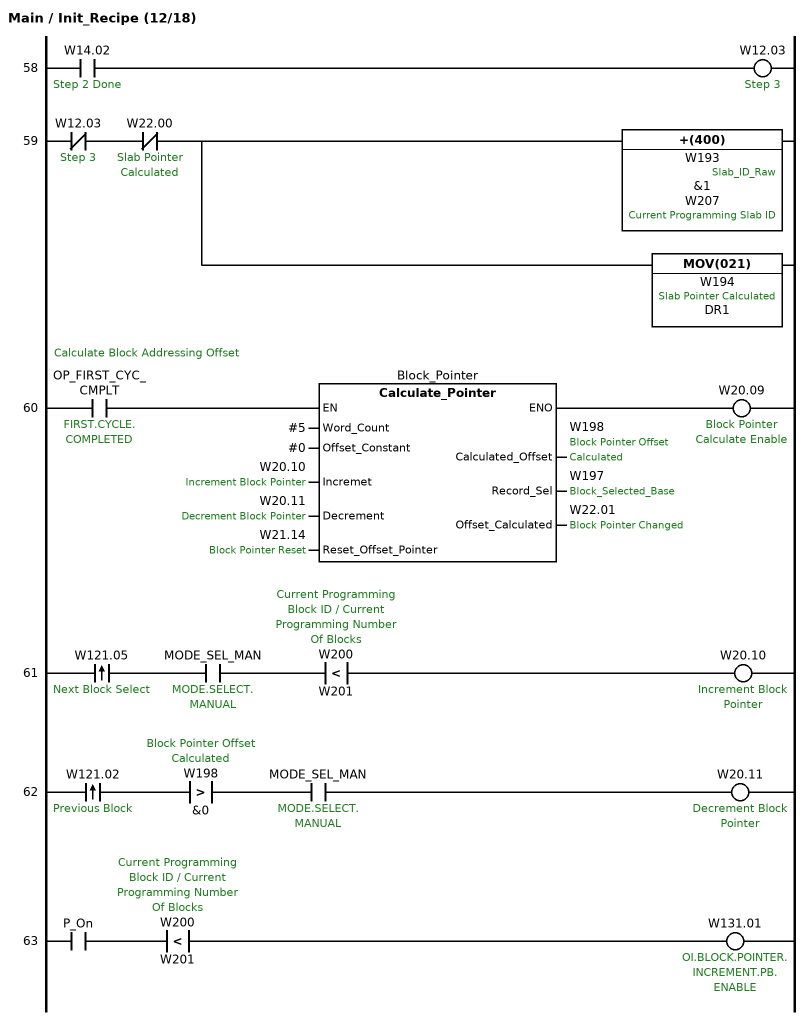
; rung 58
LD W14.02  ; Step 2 Done
OUT W12.03  ; Step 3
; rung 59
LDNOT W12.03  ; Step 3
ANDNOT W22.00  ; Slab Pointer Calculated
+(400) W193 &1 W207  ; Slab_ID_Raw, Current Programming Slab ID
MOV(021) W194 DR1  ; Slab Pointer Calculated
; rung 60: Calculate Block Addressing Offset
LD OP_FIRST_CYC_CMPLT  ; FIRST.CYCLE.COMPLETED
CALL Block_Pointer : Calculate_Pointer (Word_Count := #5, Offset_Constant := #0, Incremet := W20.10, Decrement := W20.11, Reset_Offset_Pointer := W21.14, Calculated_Offset => W198, Record_Sel => W197, Offset_Calculated => W22.01)  ; Increment Block Pointer, Decrement Block Pointer, Block Pointer Reset, Block Pointer Offset Calculated, Block_Selected_Base, Block Pointer Changed
OUT W20.09  ; Block Pointer Calculate Enable
; rung 61
@LD W121.05  ; Next Block Select
AND MODE_SEL_MAN  ; MODE.SELECT.MANUAL
AND<(310) W200 W201  ; Current Programming Block ID, Current Programming Number Of Blocks
OUT W20.10  ; Increment Block Pointer
; rung 62
@LD W121.02  ; Previous Block
AND>(320) W198 &0  ; Block Pointer Offset Calculated
AND MODE_SEL_MAN  ; MODE.SELECT.MANUAL
OUT W20.11  ; Decrement Block Pointer
; rung 63
LD P_On
AND<(310) W200 W201  ; Current Programming Block ID, Current Programming Number Of Blocks
OUT W131.01  ; OI.BLOCK.POINTER.INCREMENT.PB.ENABLE

